{attribute 'OPC.UA.DA.StructuredType':=1}
TYPE ST_RobotMoveSkill :
STRUCT
    Control     : ST_SkillControl;
    Status      : stExternalStatus;

    Specific    : ST_RobotMoveSpecific;
END_STRUCT
END_TYPE

(* stored: Version 1.1.0.1, ProductVersion 3.1.4026.18
   DUT sT_RobotMoveSkill: Id {f2feaf80-ded2-4bf9-9cb6-16352d0a1bf2} *)
